// TIA Portal V17 export
// export: Created 2023-03-06T02:05:27.4693493Z, ExportSetting WithDefaults, DisplayName Totally Integrated Automation Portal, DisplayVersion V17 Update 4, DisplayName TIA Portal Openness, DisplayVersion V17 Update 4, DisplayName TIA Portal Version Control Interface, DisplayVersion V17, DisplayName STEP 7 Professional, DisplayVersion V17 Update 4, DisplayName STEP 7 Safety, DisplayVersion V17, DisplayName WinCC Professional, DisplayVersion V17 Update 4
TYPE "PN Write"
// stored: IsFailsafeCompliant false
   STRUCT
      "x1.1" : Bool;
      "x1.2" : Bool;
      "x1.3" : Bool;
      "x1.4" : Bool;
      "x1.5" : Bool;
      "x1.6" : Bool;
      "x1.7" : Bool;
      "x1.8" : Bool;
      "x2.1" : Bool;
      "x2.2" : Bool;
      "x2.3" : Bool;
      "x2.4" : Bool;
      "x2.5" : Bool;
      "x2.6" : Bool;
      "x2.7" : Bool;
      "x2.8" : Bool;
      "x3.1" : Bool;
      "x3.2" : Bool;
      "x3.3" : Bool;
      "x3.4" : Bool;
      "x3.5" : Bool;
      "x3.6" : Bool;
      "x3.7" : Bool;
      "x3.8" : Bool;
      "x4.1" : Bool;
      "x4.2" : Bool;
      "x4.3" : Bool;
      "x4.4" : Bool;
      "x4.5" : Bool;
      "x4.6" : Bool;
      "x4.7" : Bool;
      "x4.8" : Bool;
      "x5.1" : Bool;
      "x5.2" : Bool;
      "x5.3" : Bool;
      "x5.4" : Bool;
      "x5.5" : Bool;
      "x5.6" : Bool;
      "x5.7" : Bool;
      "x5.8" : Bool;
      "x6.1" : Bool;
      "x6.2" : Bool;
      "x6.3" : Bool;
      "x6.4" : Bool;
      "x6.5" : Bool;
      "x6.6" : Bool;
      "x6.7" : Bool;
      "x6.8" : Bool;
      "x7.1" : Bool;
      "x7.2" : Bool;
      "x7.3" : Bool;
      "x7.4" : Bool;
      "x7.5" : Bool;
      "x7.6" : Bool;
      "x7.7" : Bool;
      "x7.8" : Bool;
      "x8.1" : Bool;
      "x8.2" : Bool;
      "x8.3" : Bool;
      "x8.4" : Bool;
      "x8.5" : Bool;
      "x8.6" : Bool;
      "x8.7" : Bool;
      "x8.8" : Bool;
      "x9.1" : Bool;
      "x9.2" : Bool;
      "x9.3" : Bool;
      "x9.4" : Bool;
      "x9.5" : Bool;
      "x9.6" : Bool;
      "x9.7" : Bool;
      "x9.8" : Bool;
      "x10.1" : Bool;
      "x10.2" : Bool;
      "x10.3" : Bool;
      "x10.4" : Bool;
      "x10.5" : Bool;
      "x10.6" : Bool;
      "x10.7" : Bool;
      "x10.8" : Bool;
      i1 : Int;
      i2 : Int;
      i3 : Int;
      i4 : Int;
      i5 : Int;
      i6 : Int;
      i7 : Int;
      i8 : Int;
      i9 : Int;
      i10 : Int;
      i11 : Int;
      i12 : Int;
      i13 : Int;
      i14 : Int;
      i15 : Int;
      i16 : Int;
      i17 : Int;
      i18 : Int;
      i19 : Int;
      i20 : Int;
      i21 : Int;
      i22 : Int;
      i23 : Int;
      i24 : Int;
      i25 : Int;
      i26 : Int;
      i27 : Int;
      i28 : Int;
      i29 : Int;
      i30 : Int;
      i31 : Int;
      i32 : Int;
      i33 : Int;
      i34 : Int;
      i35 : Int;
      r1 : Real;
      r2 : Real;
      r3 : Real;
      r4 : Real;
      r5 : Real;
      r6 : Real;
      r7 : Real;
      r8 : Real;
      r9 : Real;
      r10 : Real;
      r11 : Real;
      r12 : Real;
      r13 : Real;
      r14 : Real;
      r15 : Real;
      r16 : Real;
      r17 : Real;
      r18 : Real;
      r19 : Real;
      r20 : Real;
      r21 : Real;
      r22 : Real;
      r23 : Real;
      r24 : Real;
      r25 : Real;
      r26 : Real;
      r27 : Real;
      r28 : Real;
      r29 : Real;
      r30 : Real;
      r31 : Real;
      r32 : Real;
      r33 : Real;
      r34 : Real;
      r35 : Real;
      r36 : Real;
      r37 : Real;
      r38 : Real;
      r39 : Real;
      r40 : Real;
      r41 : Real;
      r42 : Real;
      r43 : Real;
      r44 : Real;
      r45 : Real;
      r46 : Real;
      r47 : Real;
      r48 : Real;
      r49 : Real;
      r50 : Real;
      r51 : Real;
      r52 : Real;
      r53 : Real;
      r54 : Real;
      r55 : Real;
      r56 : Real;
      r57 : Real;
      r58 : Real;
      r59 : Real;
      r60 : Real;
      r61 : Real;
      r62 : Real;
      r63 : Real;
      r64 : Real;
      r65 : Real;
      r66 : Real;
      r67 : Real;
      r68 : Real;
      r69 : Real;
      r70 : Real;
      r71 : Real;
      r72 : Real;
      r73 : Real;
      r74 : Real;
      r75 : Real;
      r76 : Real;
      r77 : Real;
      r78 : Real;
      r79 : Real;
      r80 : Real;
   END_STRUCT;
END_TYPE
